{attribute addProperty BoxType "EK1122-0000-0018"}
{attribute addProperty Id "Beckhoff_EPP4xxxsub_EK1100EK1100_179A0949162A_0001_EPP4174_0002_0016EPP4174_9786CACB14518.125A_0002_EPP4174_0002_0017EPP4174_9786CACB14518.125A_0003_EPP4314_1002_0016EPP4314_D38CD2FF21026.25A_0004_EPP4374_0002_0016EPP4374_6989BFFB17822.25A_0005_EPP4374_0002_0017EPP4374_6989BFFB17822.25A_0006_EPP4374_0002_0018EPP4374_6989BFFB17822.25A_0007_EPP4374_0002_0019EPP4374_6989BFFB17822.25"}
{attribute addProperty CRC "2842636463"}
{attribute addProperty SizeInBites "1228"}
{attribute addProperty SizeInBytes "153.5"}
TYPE Beckhoff_EPP4xxxEK1122_A96F30AF EXTENDS EK1122_179A0949 :
STRUCT
	{attribute addProperty Name "Beckhoff_EPP4xxxsub_EK1100"}
	Beckhoff_EPP4xxxsub_EK1100 : EK1100_179A0949;
	{attribute addProperty Name "A_0001_EPP4174_0002_0016"}
	A_0001_EPP4174_0002_0016 : EPP4174_9786CACB;
	{attribute addProperty Name "A_0002_EPP4174_0002_0017"}
	A_0002_EPP4174_0002_0017 : EPP4174_9786CACB;
	{attribute addProperty Name "A_0003_EPP4314_1002_0016"}
	A_0003_EPP4314_1002_0016 : EPP4314_D38CD2FF;
	{attribute addProperty Name "A_0004_EPP4374_0002_0016"}
	A_0004_EPP4374_0002_0016 : EPP4374_6989BFFB;
	{attribute addProperty Name "A_0005_EPP4374_0002_0017"}
	A_0005_EPP4374_0002_0017 : EPP4374_6989BFFB;
	{attribute addProperty Name "A_0006_EPP4374_0002_0018"}
	A_0006_EPP4374_0002_0018 : EPP4374_6989BFFB;
	{attribute addProperty Name "A_0007_EPP4374_0002_0019"}
	A_0007_EPP4374_0002_0019 : EPP4374_6989BFFB;
END_STRUCT
END_TYPE

(* stored: Version 1.2.0.0, ProductVersion 3.1.4024.9
   DUT Beckhoff_EPP4xxxEK1122_A96F30AF: Id {7d7b8b3c-efbf-4eaa-9e01-c0657412c033} *)
